           // Deciding which Position
           // Position - Belt
           IF "gtyp_Setup".i_Pos_Selection = 21 THEN
               #ldi_Pos_Horizontal := "gtyp_HBW".di_PosBelt_Horizontal;
               #ldi_Pos_Vertical := "gtyp_HBW".di_PosBelt_Vertical;
               #ldi_Offset_Vertical := "gtyp_HBW".di_Offset_Pos_Belt_Vertical;
               // Position - A1 
           ELSIF "gtyp_Setup".i_Pos_Selection = 22 THEN
               #ldi_Pos_Horizontal := "gtyp_HBW".di_PosRack_A1_Horizontal;
               #ldi_Pos_Vertical := "gtyp_HBW".di_PosRack_A1_Vertical;
               #ldi_Offset_Vertical := "gtyp_HBW".di_Offset_Pos_Rack_Vertical;
               // Position - B2 
           ELSIF "gtyp_Setup".i_Pos_Selection = 23 THEN
               #ldi_Pos_Horizontal := "gtyp_HBW".di_PosRack_B2_Horizontal;
               #ldi_Pos_Vertical := "gtyp_HBW".di_PosRack_B2_Vertical;
               #ldi_Offset_Vertical := "gtyp_HBW".di_Offset_Pos_Rack_Vertical;
               // Position - C3 
           ELSIF "gtyp_Setup".i_Pos_Selection = 24 THEN
               #ldi_Pos_Horizontal := "gtyp_HBW".di_PosRack_C3_Horizontal;
               #ldi_Pos_Vertical := "gtyp_HBW".di_PosRack_C3_Vertical;
               #ldi_Offset_Vertical := "gtyp_HBW".di_Offset_Pos_Rack_Vertical;
           END_IF;
       END_IF;

       // Set Positioning activ?
       IF NOT "gtyp_Setup".x_Set_Pos_Activ THEN
           "gtyp_Setup".i_Pos_Selection := 0;
       END_IF;

       // step chain HBW
       CASE #li_StepCase OF

           0:  // init
               #lx_Start_TON_Wait := FALSE;
               #li_StepCase := 10;

           10:  // Set Positioning activ?
               IF "gtyp_Setup".x_Set_Pos_Activ
                   AND (("gtyp_Setup".i_Pos_Selection > 20)
                   AND ("gtyp_Setup".i_Pos_Selection < 41)) THEN

                   "gtyp_HBW".Horizontal_Axis.x_Start_Positioning := FALSE;
                   "gtyp_HBW".Vertical_Axis.x_Start_Positioning := FALSE;
                   "gtyp_HBW".Horizontal_Axis.x_Reference := FALSE;
                   "gtyp_HBW".Vertical_Axis.x_Reference := FALSE;
                   "gtyp_Setup".x_Start_Positioning := FALSE;
                   "gtyp_Setup".x_Final_Positioning := FALSE;
                   "gtyp_Setup".x_Home_Positioning := FALSE;
                   "gtyp_Setup".x_Start_Offset := FALSE;
                   "QX_HBW_M4_CantileverBackward_Q8" := FALSE;
                   "QX_HBW_M4_CantileverForward_Q7" := FALSE;
                   #li_StepCase := 20;
               END_IF;

           20: //homing vertical/horizontal axis

               "gtyp_HBW".Horizontal_Axis.x_Reference := TRUE;
               "gtyp_HBW".Vertical_Axis.x_Reference := TRUE;

               IF NOT "gtyp_HBW".Horizontal_Axis.x_Referenced AND NOT "gtyp_HBW".Vertical_Axis.x_Referenced THEN
                   #li_StepCase := 30;
               END_IF;

           30: // homed vertical/horizontal axis
               IF "gtyp_HBW".Horizontal_Axis.x_Referenced THEN
                   "gtyp_HBW".Horizontal_Axis.x_Reference := FALSE;
               END_IF;
               IF "gtyp_HBW".Vertical_Axis.x_Referenced THEN
                   "gtyp_HBW".Vertical_Axis.x_Reference := FALSE;
               END_IF;

               IF "gtyp_HBW".Horizontal_Axis.x_Referenced AND "gtyp_HBW".Vertical_Axis.x_Referenced THEN
                   "gtyp_HBW".Horizontal_Axis.x_Reference := FALSE;
                   "gtyp_HBW".Vertical_Axis.x_Reference := FALSE;
                   #li_StepCase := 40;
               END_IF;

           40: // Start Positioning Step next
               IF "gtyp_Setup".x_Start_Positioning OR #lx_Start_Positioning_m OR #lx_Start_FinalPositioning_m OR #lx_Start_Offset_m THEN
                   #lx_Start_Positioning_m := FALSE;
                   #li_StepCase := 50;
               END_IF;

           50: // Position vertical/horizontal HBW
               "gtyp_HBW".Horizontal_Axis.di_Target_Position := #ldi_Pos_Horizontal;
               "gtyp_HBW".Horizontal_Axis.x_Start_Positioning := TRUE;
               "gtyp_HBW".Vertical_Axis.di_Target_Position := #ldi_Pos_Vertical;
               "gtyp_HBW".Vertical_Axis.x_Start_Positioning := TRUE;

               IF ("gtyp_HBW".Horizontal_Axis.di_Actual_Position <= (#ldi_Pos_Horizontal + "gtyp_HBW".Horizontal_Axis.Config.di_Pos_Window))
                   AND ("gtyp_HBW".Horizontal_Axis.di_Actual_Position >= (#ldi_Pos_Horizontal - "gtyp_HBW".Horizontal_Axis.Config.di_Pos_Window))
                   AND "gtyp_HBW".Horizontal_Axis.x_Position_Reached THEN
                   "gtyp_HBW".Horizontal_Axis.x_Start_Positioning := FALSE;
               END_IF;

               IF ("gtyp_HBW".Vertical_Axis.di_Actual_Position <= (#ldi_Pos_Vertical + "gtyp_HBW".Vertical_Axis.Config.di_Pos_Window))
                   AND ("gtyp_HBW".Vertical_Axis.di_Actual_Position >= (#ldi_Pos_Vertical - "gtyp_HBW".Vertical_Axis.Config.di_Pos_Window))
                   AND "gtyp_HBW".Vertical_Axis.x_Position_Reached THEN
                   "gtyp_HBW".Vertical_Axis.x_Start_Positioning := FALSE;
               END_IF;

               IF ("gtyp_HBW".Horizontal_Axis.di_Actual_Position <= (#ldi_Pos_Horizontal + "gtyp_HBW".Horizontal_Axis.Config.di_Pos_Window))
                   AND ("gtyp_HBW".Horizontal_Axis.di_Actual_Position >= (#ldi_Pos_Horizontal - "gtyp_HBW".Horizontal_Axis.Config.di_Pos_Window))
                   AND "gtyp_HBW".Horizontal_Axis.x_Position_Reached
                   AND ("gtyp_HBW".Vertical_Axis.di_Actual_Position <= (#ldi_Pos_Vertical + "gtyp_HBW".Vertical_Axis.Config.di_Pos_Window))
                   AND ("gtyp_HBW".Vertical_Axis.di_Actual_Position >= (#ldi_Pos_Vertical - "gtyp_HBW".Vertical_Axis.Config.di_Pos_Window))
                   AND "gtyp_HBW".Vertical_Axis.x_Position_Reached THEN
                   "gtyp_HBW".Horizontal_Axis.x_Start_Positioning := FALSE;
                   "gtyp_HBW".Vertical_Axis.x_Start_Positioning := FALSE;
                   "gtyp_Setup".x_Start_Positioning := FALSE;
                   #li_StepCase := 60;
               END_IF;

           60: // Deciding which doing

               // Start new Positioning
               IF "gtyp_Setup".x_Start_Positioning THEN
                   #lx_Start_Positioning_m := TRUE;
                   #li_StepCase := 10;
                   // Start Final Positioning
               ELSIF "gtyp_Setup".x_Final_Positioning OR #lx_Start_FinalPositioning_m OR #lx_Start_Offset_m THEN
                   #lx_Start_FinalPositioning_m := FALSE;
                   #li_StepCase := 70;
                   // Deaktivate Set Positioning
               ELSIF #lfb_R_Trig_Deaktivate.Q OR "gtyp_Setup".x_Home_Positioning THEN
                   "gtyp_Setup".x_Home_Positioning := FALSE;
                   #li_StepCase := 110;
               END_IF;

           70: // Final Positioning - Cantilever Forward

               "QX_HBW_M4_CantileverBackward_Q8" := FALSE;
               "QX_HBW_M4_CantileverForward_Q7" := TRUE;

               IF "IX_HBW_SwitchCantileverFront_I5" AND NOT "IX_HBW_SwitchCantileverBack_I6" THEN
                   "QX_HBW_M4_CantileverBackward_Q8" := FALSE;
                   "QX_HBW_M4_CantileverForward_Q7" := FALSE;
                   "gtyp_Setup".x_Final_Positioning := FALSE;
                   #li_StepCase := 80;
               END_IF;

           80: // Deciding which doing

               // Start new Positioning
               IF "gtyp_Setup".x_Start_Positioning THEN
                   #lx_Start_Positioning_m := TRUE;
                   #li_StepCase := 110;
                   // Start Final Positioning
               ELSIF "gtyp_Setup".x_Final_Positioning THEN
                   #lx_Start_FinalPositioning_m := TRUE;
                   #li_StepCase := 110;
                   // Start Final Positioning
               ELSIF "gtyp_Setup".x_Start_Offset OR #lx_Start_Offset_m THEN
                   #lx_Start_Offset_m := FALSE;
                   #li_StepCase := 90;
                   // Deaktivate Set Positioning
               ELSIF #lfb_R_Trig_Deaktivate.Q OR "gtyp_Setup".x_Home_Positioning THEN
                   "gtyp_Setup".x_Home_Positioning := FALSE;
                   #li_StepCase := 110;
               END_IF;

           90: // Position vertical+offset HBW
               "gtyp_HBW".Vertical_Axis.di_Target_Position := #ldi_Pos_Vertical - #ldi_Offset_Vertical;
               "gtyp_HBW".Vertical_Axis.x_Start_Positioning := TRUE;

               IF ("gtyp_HBW".Vertical_Axis.di_Actual_Position <= (#ldi_Pos_Vertical - #ldi_Offset_Vertical + "gtyp_HBW".Vertical_Axis.Config.di_Pos_Window))
                   AND ("gtyp_HBW".Vertical_Axis.di_Actual_Position >= (#ldi_Pos_Vertical - #ldi_Offset_Vertical - "gtyp_HBW".Vertical_Axis.Config.di_Pos_Window))
                   AND "gtyp_HBW".Vertical_Axis.x_Position_Reached THEN
                   "gtyp_HBW".Vertical_Axis.x_Start_Positioning := FALSE;
                   "gtyp_Setup".x_Start_Offset := FALSE;
                   #li_StepCase := 100;
               END_IF;

           100: // Deciding which doing

               // Start new Positioning
               IF "gtyp_Setup".x_Start_Positioning THEN
                   #lx_Start_Positioning_m := TRUE;
                   #li_StepCase := 110;
                   // Start Final Positioning
               ELSIF "gtyp_Setup".x_Final_Positioning THEN
                   #lx_Start_FinalPositioning_m := TRUE;
                   #li_StepCase := 110;
                   // Start Final Positioning
               ELSIF "gtyp_Setup".x_Start_Offset THEN
                   #lx_Start_Offset_m := true;
                   #li_StepCase := 110;
                   // Deaktivate Set Positioning
               ELSIF #lfb_R_Trig_Deaktivate.Q OR "gtyp_Setup".x_Home_Positioning THEN
                   "gtyp_Setup".x_Home_Positioning := FALSE;
                   #li_StepCase := 110;
               END_IF;

           110: // Position vertical HBW
               "gtyp_HBW".Vertical_Axis.di_Target_Position := #ldi_Pos_Vertical;
               "gtyp_HBW".Vertical_Axis.x_Start_Positioning := TRUE;

               IF ("gtyp_HBW".Vertical_Axis.di_Actual_Position <= (#ldi_Pos_Vertical + "gtyp_HBW".Vertical_Axis.Config.di_Pos_Window))
                   AND ("gtyp_HBW".Vertical_Axis.di_Actual_Position >= (#ldi_Pos_Vertical - "gtyp_HBW".Vertical_Axis.Config.di_Pos_Window))
                   AND "gtyp_HBW".Vertical_Axis.x_Position_Reached THEN
                   "gtyp_HBW".Vertical_Axis.x_Start_Positioning := FALSE;
                   #li_StepCase := 120;
               END_IF;

           120: // Position vertical Back HBW

               "QX_HBW_M4_CantileverBackward_Q8" := TRUE;
               "QX_HBW_M4_CantileverForward_Q7" := FALSE;

               IF NOT "IX_HBW_SwitchCantileverFront_I5" AND "IX_HBW_SwitchCantileverBack_I6" THEN
                   "QX_HBW_M4_CantileverBackward_Q8" := FALSE;
                   "QX_HBW_M4_CantileverForward_Q7" := FALSE;
                   #li_StepCase := 130;
               END_IF;

           130: // homing vertical/horizontal axis

               "gtyp_HBW".Horizontal_Axis.x_Reference := TRUE;
               "gtyp_HBW".Vertical_Axis.x_Reference := TRUE;

               IF NOT "gtyp_HBW".Horizontal_Axis.x_Referenced AND NOT "gtyp_HBW".Vertical_Axis.x_Referenced THEN
                   #li_StepCase := 140;
               END_IF;

           140: //homed vertical/horizontal axis
               IF "gtyp_HBW".Horizontal_Axis.x_Referenced THEN
                   "gtyp_HBW".Horizontal_Axis.x_Reference := FALSE;
               END_IF;
               IF "gtyp_HBW".Vertical_Axis.x_Referenced THEN
                   "gtyp_HBW".Vertical_Axis.x_Reference := FALSE;
               END_IF;

               IF "gtyp_HBW".Horizontal_Axis.x_Referenced AND "gtyp_HBW".Vertical_Axis.x_Referenced THEN
                   "gtyp_HBW".Horizontal_Axis.x_Reference := FALSE;
                   "gtyp_HBW".Vertical_Axis.x_Reference := FALSE;
                   #li_StepCase := 0;
               END_IF;

               // Statement section ELSE    
           ELSE
               ;
       END_CASE;

       IF (("gtyp_Setup".i_Pos_Selection > 20)
           AND ("gtyp_Setup".i_Pos_Selection < 41)) THEN
           // Reload Pos Value
           "gtyp_Setup".di_Pos_Horizontal := #ldi_Pos_Horizontal;
           "gtyp_Setup".di_Pos_Vertical := #ldi_Pos_Vertical;
           "gtyp_Setup".di_Pos_Rotate := 0;
       END_IF;
   ELSE
       #lx_Init := TRUE;
   END_IF;
END_FUNCTION_BLOCK

FUNCTION_BLOCK "PRG_SSC_Calibration_Color"   // FB32, SCL
TITLE = Program Calibration Color Sensor SSC
{ S7_Optimized_Access := 'TRUE' }
AUTHOR : A.Schaefer
VERSION : 0.0
   VAR
      lx_Init : Bool;
      lx_Start_TON_Wait : Bool;
      lx_Start_Positioning_m : Bool;
      lt_TON_Wait : Time;
      li_StepCase : Int;
      ldi_Pos_Horizontal : DInt;
      ldi_Pos_Vertical : DInt;
      lfb_R_Trig_Deaktivate : R_TRIG;
      lfb_TON_Wait : TON_TIME;
   END_VAR
BEGIN
   IF #lx_Init THEN

       // FB TON Wait
       #lfb_TON_Wait(IN := #lx_Start_TON_Wait,
                     PT := #lt_TON_Wait);

       #lfb_R_Trig_Deaktivate(CLK := NOT "gtyp_Setup".x_Color_Sensor_Calibration
                              OR NOT ("gtyp_Setup".i_Color_Sensor_Selection = 1));
       // Deaktivate step 0   
       IF #lfb_R_Trig_Deaktivate.Q THEN
           "gtyp_Setup".x_Calculate_Value_Color := FALSE;
           "gtyp_Setup".x_Set_Calib_Value_Color_Blue := FALSE;
           "gtyp_Setup".x_Set_Calib_Value_Color_Red := FALSE;
           "gtyp_Setup".x_Set_Calib_Value_Color_White := FALSE;
           "gtyp_Setup".w_Calib_ColorValue_Blue := 0;
           "gtyp_Setup".w_Calib_ColorValue_Red := 0;
           "gtyp_Setup".w_Calib_ColorValue_White := 0;
           "gtyp_Setup".w_Threshold_Red_Blue := 0;
           "gtyp_Setup".w_Threshold_White_Red := 0;
           #li_StepCase := 0;
       END_IF;

       // step chain HBW
       CASE #li_StepCase OF

           0:  // init
               #lx_Start_TON_Wait := FALSE;
               #li_StepCase := 10;

           10:  // Set Calibration activ?
               IF "gtyp_Setup".x_Color_Sensor_Calibration
                   AND ("gtyp_Setup".i_Color_Sensor_Selection = 1) THEN
                   "gtyp_Setup".x_Calculate_Value_Color := FALSE;
                   "gtyp_Setup".x_Set_Calib_Value_Color_Blue := FALSE;
                   "gtyp_Setup".x_Set_Calib_Value_Color_Red := FALSE;
                   "gtyp_Setup".x_Set_Calib_Value_Color_White := FALSE;
                   "gtyp_Setup".w_Calib_ColorValue_Blue := 0;
                   "gtyp_Setup".w_Calib_ColorValue_Red := 0;
                   "gtyp_Setup".w_Calib_ColorValue_White := 0;
                   "gtyp_Setup".w_Threshold_Red_Blue := 0;
                   "gtyp_Setup".w_Threshold_White_Red := 0;
                   #li_StepCase := 20;
               END_IF;

           20: // wait for set Values or Calculate

               // Start new Positioning
               IF "gtyp_Setup".x_Set_Calib_Value_Color_Blue THEN
                   "gtyp_Setup".w_Calib_ColorValue_Blue := "IW_SSC_ColorSensor_A1";
                   "gtyp_Setup".x_Set_Calib_Value_Color_Blue := FALSE;
               ELSIF "gtyp_Setup".x_Set_Calib_Value_Color_Red THEN
                   "gtyp_Setup".w_Calib_ColorValue_Red := "IW_SSC_ColorSensor_A1";
                   "gtyp_Setup".x_Set_Calib_Value_Color_Red := FALSE;
               ELSIF "gtyp_Setup".x_Set_Calib_Value_Color_White THEN
                   "gtyp_Setup".w_Calib_ColorValue_White := "IW_SSC_ColorSensor_A1";
                   "gtyp_Setup".x_Set_Calib_Value_Color_White := FALSE;
               END_IF;

               "gtyp_Setup".w_Threshold_White_Red := "gtyp_Setup".w_Calib_ColorValue_White + (("gtyp_Setup".w_Calib_ColorValue_Red - "gtyp_Setup".w_Calib_ColorValue_White) / 2);
               "gtyp_Setup".w_Threshold_Red_Blue := "gtyp_Setup".w_Calib_ColorValue_Red + (("gtyp_Setup".w_Calib_ColorValue_Blue - "gtyp_Setup".w_Calib_ColorValue_Red) / 2);

               IF "gtyp_Setup".x_Calculate_Value_Color THEN
                   "gtyp_SSC".w_Threshold_White_Red := "gtyp_Setup".w_Threshold_White_Red;
                   "gtyp_SSC".w_Threshold_Red_Blue := "gtyp_Setup".w_Threshold_Red_Blue;
                   "gtyp_Setup".x_Calculate_Value_Color := FALSE;
               END_IF;

               // Statement section ELSE    
           ELSE
               ;
       END_CASE;

       IF ("gtyp_Setup".i_Color_Sensor_Selection = 1) THEN
           // Reload Pos Value
           "gtyp_Setup".w_Actual_ColorValue := "IW_SSC_ColorSensor_A1";
       END_IF;
   ELSE
       #lx_Init := TRUE;
   END_IF;
END_FUNCTION_BLOCK

FUNCTION_BLOCK "PRG_SLD_Calibration_Color"   // FB33, SCL
TITLE = Program Calibration Color Sensor SLD
{ S7_Optimized_Access := 'TRUE' }
AUTHOR : A.Schaefer
VERSION : 0.0
   VAR
      lx_Init : Bool;
      lx_Start_TON_Wait : Bool;
      lx_Start_Positioning_m : Bool;
      lt_TON_Wait : Time;
      li_StepCase : Int;
      lw_ColorValueMin : Word;
      ldi_Pos_Horizontal : DInt;
      ldi_Pos_Vertical : DInt;
      lfb_R_Trig_Deaktivate : R_TRIG;
      lfb_TON_Wait : TON_TIME;
   END_VAR
BEGIN
   IF #lx_Init THEN

       // FB TON Wait
       #lfb_TON_Wait(IN := #lx_Start_TON_Wait,
                     PT := #lt_TON_Wait);

       #lfb_R_Trig_Deaktivate(CLK := NOT "gtyp_Setup".x_Color_Sensor_Calibration
                              OR NOT ("gtyp_Setup".i_Color_Sensor_Selection = 2));
       // Deaktivate step 0   
       IF #lfb_R_Trig_Deaktivate.Q THEN
           "gtyp_Setup".x_Calculate_Value_Color := FALSE;
           "gtyp_Setup".x_Set_Calib_Value_Color_Blue := FALSE;
           "gtyp_Setup".x_Set_Calib_Value_Color_Red := FALSE;
           "gtyp_Setup".x_Set_Calib_Value_Color_White := FALSE;
           "gtyp_Setup".w_Calib_ColorValue_Blue := 0;
           "gtyp_Setup".w_Calib_ColorValue_Red := 0;
           "gtyp_Setup".w_Calib_ColorValue_White := 0;
           "gtyp_Setup".w_Threshold_Red_Blue := 0;
           "gtyp_Setup".w_Threshold_White_Red := 0;
           "QX_SLD_M1_ConveyorBelt_Q1" := FALSE;
           #lw_ColorValueMin := 16#FF;
           #li_StepCase := 0;
       END_IF;

       // step chain HBW
       CASE #li_StepCase OF

           0:  // init
               #lx_Start_TON_Wait := FALSE;
               #li_StepCase := 10;

           10:  // Set Calibration activ?
               IF "gtyp_Setup".x_Color_Sensor_Calibration
                   AND ("gtyp_Setup".i_Color_Sensor_Selection = 2) THEN
                   "gtyp_Setup".x_Calculate_Value_Color := FALSE;
                   "gtyp_Setup".x_Set_Calib_Value_Color_Blue := FALSE;
                   "gtyp_Setup".x_Set_Calib_Value_Color_Red := FALSE;
                   "gtyp_Setup".x_Set_Calib_Value_Color_White := FALSE;
                   "gtyp_Setup".w_Calib_ColorValue_Blue := 0;
                   "gtyp_Setup".w_Calib_ColorValue_Red := 0;
                   "gtyp_Setup".w_Calib_ColorValue_White := 0;
                   "gtyp_Setup".w_Threshold_Red_Blue := 0;
                   "gtyp_Setup".w_Threshold_White_Red := 0;
                   "QX_SLD_M1_ConveyorBelt_Q1" := FALSE;
                   #lw_ColorValueMin := 16#FFFF;
                   #li_StepCase := 20;
               END_IF;

           20: // wait for set Values or Calculate

               IF NOT "IX_SLD_LightBarrierInlet_I2" THEN
                   "QX_SLD_M1_ConveyorBelt_Q1" := TRUE;
                   #lw_ColorValueMin := 16#FFFF;
               END_IF;

               IF #lw_ColorValueMin > "IW_SLD_ColorSensor_A4" THEN
                   #lw_ColorValueMin := "IW_SLD_ColorSensor_A4";
               END_IF;

               IF NOT "IX_SLD_LightBarrierBehindColorSensor_I3" THEN
                   "QX_SLD_M1_ConveyorBelt_Q1" := FALSE;
               END_IF;

               // Start new Positioning
               IF "gtyp_Setup".x_Set_Calib_Value_Color_Blue THEN
                   "gtyp_Setup".w_Calib_ColorValue_Blue := #lw_ColorValueMin;
                   "gtyp_Setup".x_Set_Calib_Value_Color_Blue := FALSE;
               ELSIF "gtyp_Setup".x_Set_Calib_Value_Color_Red THEN
                   "gtyp_Setup".w_Calib_ColorValue_Red := #lw_ColorValueMin;
                   "gtyp_Setup".x_Set_Calib_Value_Color_Red := FALSE;
               ELSIF "gtyp_Setup".x_Set_Calib_Value_Color_White THEN
                   "gtyp_Setup".w_Calib_ColorValue_White := #lw_ColorValueMin;
                   "gtyp_Setup".x_Set_Calib_Value_Color_White := FALSE;
               END_IF;

               "gtyp_Setup".w_Threshold_White_Red := "gtyp_Setup".w_Calib_ColorValue_White + (("gtyp_Setup".w_Calib_ColorValue_Red - "gtyp_Setup".w_Calib_ColorValue_White) / 2);
               "gtyp_Setup".w_Threshold_Red_Blue := "gtyp_Setup".w_Calib_ColorValue_Red + (("gtyp_Setup".w_Calib_ColorValue_Blue - "gtyp_Setup".w_Calib_ColorValue_Red) / 2);

               IF "gtyp_Setup".x_Calculate_Value_Color THEN
                   "gtyp_SLD".w_Threshold_White_Red := "gtyp_Setup".w_Threshold_White_Red;
                   "gtyp_SLD".w_Threshold_Red_Blue := "gtyp_Setup".w_Threshold_Red_Blue;
                   "gtyp_Setup".x_Calculate_Value_Color := FALSE;
               END_IF;

               // Statement section ELSE    
           ELSE
               ;
       END_CASE;

       IF ("gtyp_Setup".i_Color_Sensor_Selection = 2) THEN
           // Reload Pos Value
           "gtyp_Setup".w_Actual_ColorValue := "IW_SLD_ColorSensor_A4";
       END_IF;
   ELSE
       #lx_Init := TRUE;
   END_IF;
END_FUNCTION_BLOCK

FUNCTION_BLOCK "PRG_SLD_Set_Counter_Values"   // FB34, SCL
TITLE = Program Set counter Values SLD
{ S7_Optimized_Access := 'TRUE' }
AUTHOR : A.Schaefer
VERSION : 0.0
   VAR
      lx_Init : Bool;
      lfb_R_Trig_Calib_activ : R_TRIG;
   END_VAR
BEGIN
   IF #lx_Init THEN

       // Reload act. Counter Values
       IF NOT "gtyp_Setup".x_Counter_Value_Calibration THEN
           "gtyp_Setup".i_Calib_CounterValue_Blue := "gtyp_SLD".i_CounterValue_Blue;
           "gtyp_Setup".i_Calib_CounterValue_Red := "gtyp_SLD".i_CounterValue_Red;
           "gtyp_Setup".i_Calib_CounterValue_White := "gtyp_SLD".i_CounterValue_White;
       END_IF;

       // Set Counter Values   
       IF "gtyp_Setup".x_Set_CounterValues AND "gtyp_Setup".x_Counter_Value_Calibration THEN
           "gtyp_SLD".i_CounterValue_Blue := "gtyp_Setup".i_Calib_CounterValue_Blue;
           "gtyp_SLD".i_CounterValue_Red := "gtyp_Setup".i_Calib_CounterValue_Red;
           "gtyp_SLD".i_CounterValue_White := "gtyp_Setup".i_Calib_CounterValue_White;
           "gtyp_Setup".x_Set_CounterValues := FALSE;
       END_IF;

   ELSE
       #lx_Init := TRUE;
   END_IF;
END_FUNCTION_BLOCK

FUNCTION_BLOCK "PRG_VGR_Set_Park_Position"   // FB35, SCL
TITLE = Program Set Positioning VGR
{ S7_Optimized_Access := 'TRUE' }
AUTHOR : A.Schaefer
VERSION : 0.0
   VAR
      lx_Init : Bool;
      lx_Start_TON_Wait : Bool;
      lt_TON_Wait : Time;
      li_StepCase : Int;
      lfb_TON_Wait : TON_TIME;
      lfb_R_Trig_Start_Park_Pos : R_TRIG;
   END_VAR
BEGIN
   IF #lx_Init THEN

       // FB TON Wait
       #lfb_TON_Wait(IN := #lx_Start_TON_Wait,
                     PT := #lt_TON_Wait);

       #lfb_R_Trig_Start_Park_Pos(CLK := "gtyp_Setup".x_Park_Position
                                  OR "IX_Set_Park_Position");

       // Set Start Park Position   
       IF #lfb_R_Trig_Start_Park_Pos.Q THEN
           "gtyp_VGR".x_Start_Park_Position := TRUE;
           #li_StepCase := 0;
       END_IF;

       // not Start Park Pos Step 0
       IF NOT "gtyp_VGR".x_Start_Park_Position THEN
           #li_StepCase := 0;
       END_IF;

       // step chain HBW
       CASE #li_StepCase OF

           0:  // init
               #lx_Start_TON_Wait := FALSE;
               #li_StepCase := 10;

           10:  // Set Positioning activ?
               IF "gtyp_VGR".x_Start_Park_Position AND NOT "gtyp_VGR".x_Park_Position_Reached THEN
                   "gtyp_VGR".horizontal_Axis.x_Start_Positioning := FALSE;
                   "gtyp_VGR".vertical_Axis.x_Start_Positioning := FALSE;
                   "gtyp_VGR".rotate_Axis.x_Start_Positioning := FALSE;
                   "gtyp_VGR".horizontal_Axis.x_Reference := FALSE;
                   "gtyp_VGR".vertical_Axis.x_Reference := FALSE;
                   "gtyp_VGR".rotate_Axis.x_Reference := FALSE;
                   "gtyp_VGR".vertical_Axis.i_PWM := 800;
                   #li_StepCase := 20;
               END_IF;

           20: // homing vertical axis
               "gtyp_VGR".vertical_Axis.x_Reference := TRUE;

               IF NOT "gtyp_VGR".vertical_Axis.x_Referenced THEN
                   #li_StepCase := 30;
               END_IF;

           30: // homed vertical axis
               IF "gtyp_VGR".vertical_Axis.x_Referenced THEN
                   "gtyp_VGR".vertical_Axis.x_Reference := FALSE;
                   #li_StepCase := 40;
               END_IF;

           40: // homing horizontal axis
               "gtyp_VGR".horizontal_Axis.x_Reference := TRUE;

               IF NOT "gtyp_VGR".horizontal_Axis.x_Referenced THEN
                   #li_StepCase := 50;
               END_IF;

           50: // homed horizontal axis
               IF "gtyp_VGR".horizontal_Axis.x_Referenced THEN
                   "gtyp_VGR".horizontal_Axis.x_Reference := FALSE;
                   #li_StepCase := 60;
               END_IF;

           60: // homing rotate axis
               "gtyp_VGR".rotate_Axis.x_Reference := TRUE;

               IF NOT "gtyp_VGR".rotate_Axis.x_Referenced THEN
                   #li_StepCase := 70;
               END_IF;

           70: // homed rotate axis
               IF "gtyp_VGR".rotate_Axis.x_Referenced THEN
                   "gtyp_VGR".rotate_Axis.x_Reference := FALSE;
                   #li_StepCase := 80;
               END_IF;

           80: // Position rotate Axis
               "gtyp_VGR".rotate_Axis.di_Target_Position := "gtyp_VGR".di_Pos_Park_rotate;
               "gtyp_VGR".rotate_Axis.x_Start_Positioning := TRUE;

               IF ("gtyp_VGR".rotate_Axis.di_Actual_Position <= ("gtyp_VGR".di_Pos_Park_rotate + "gtyp_VGR".rotate_Axis.Config.di_Pos_Window))
                   AND ("gtyp_VGR".rotate_Axis.di_Actual_Position >= ("gtyp_VGR".di_Pos_Park_rotate - "gtyp_VGR".rotate_Axis.Config.di_Pos_Window))
                   AND "gtyp_VGR".rotate_Axis.x_Position_Reached THEN
                   "gtyp_VGR".rotate_Axis.x_Start_Positioning := FALSE;
                   #li_StepCase := 90;
               END_IF;

           90: // Position horizontal Axis
               "gtyp_VGR".horizontal_Axis.di_Target_Position := "gtyp_VGR".di_Pos_Park_horizontal;
               "gtyp_VGR".horizontal_Axis.x_Start_Positioning := TRUE;

               IF ("gtyp_VGR".horizontal_Axis.di_Actual_Position <= ("gtyp_VGR".di_Pos_Park_horizontal + "gtyp_VGR".horizontal_Axis.Config.di_Pos_Window))
                   AND ("gtyp_VGR".horizontal_Axis.di_Actual_Position >= ("gtyp_VGR".di_Pos_Park_horizontal - "gtyp_VGR".horizontal_Axis.Config.di_Pos_Window))
                   AND "gtyp_VGR".horizontal_Axis.x_Position_Reached THEN
                   "gtyp_VGR".horizontal_Axis.x_Start_Positioning := FALSE;
                   #li_StepCase := 100;
               END_IF;

           100: // Position vertical Axis
               "gtyp_VGR".vertical_Axis.i_PWM := 500;
               "gtyp_VGR".vertical_Axis.di_Target_Position := "gtyp_VGR".di_Pos_Park_vertical;
               "gtyp_VGR".vertical_Axis.x_Start_Positioning := TRUE;

               IF ("gtyp_VGR".vertical_Axis.di_Actual_Position <= ("gtyp_VGR".di_Pos_Park_vertical + "gtyp_VGR".vertical_Axis.Config.di_Pos_Window))
                   AND ("gtyp_VGR".vertical_Axis.di_Actual_Position >= ("gtyp_VGR".di_Pos_Park_vertical - "gtyp_VGR".vertical_Axis.Config.di_Pos_Window))
                   AND "gtyp_VGR".vertical_Axis.x_Position_Reached THEN
                   "gtyp_VGR".vertical_Axis.x_Start_Positioning := FALSE;
                   #li_StepCase := 110;
               END_IF;

           110: // Deciding which doing
               "gtyp_VGR".x_Park_Position_Reached := TRUE;


               // Statement section ELSE    
           ELSE
               ;
       END_CASE;

   ELSE
       #lx_Init := TRUE;
   END_IF;
END_FUNCTION_BLOCK

FUNCTION_BLOCK "PRG_DSO_Status"   // FB36, SCL
TITLE = Program Status DSO
{ S7_Optimized_Access := 'TRUE' }
AUTHOR : A.Schaefer
VERSION : 0.0
   VAR
      lx_Init : Bool;
      lx_Start : Bool;
      li_StepCase : Int;
      ldt_MQTT : Date_And_Time;
      li_Return_LDT : Int;
      li_code_old : Int;
      lfb_R_Trig_Outsourcing : R_TRIG;
      lfb_R_Trig_Take_Workpiece : R_TRIG;
      lfb_TON_Status : TON_TIME;
      lfb_TON_End_Order : TON_TIME;
      lx_StartStatus : Bool;
      lx_StartEndOrder : Bool;
      lx_StartTimer : Bool;
   END_VAR
BEGIN
   IF #lx_Init THEN

       // wait time state
       #lfb_TON_Status(IN := NOT #lx_StartStatus,
                       PT := T#2s);

       // rising/falling edge light barrier DSI
       #lfb_R_Trig_Outsourcing(CLK := NOT "IX_SSC_LightBarrierOutsourcing_I4");
       #lfb_R_Trig_Take_Workpiece(CLK := "IX_SSC_LightBarrierOutsourcing_I4");

       // start wait time end order 
       IF NOT "IX_SSC_LightBarrierOutsourcing_I4" AND ("gtyp_Interface_Dashboard".Subscribe.State_Order.s_state = 'SHIPPED') THEN
           #lx_StartEndOrder := TRUE;
       END_IF;

       // wait time end order
       #lfb_TON_End_Order(IN := #lx_StartEndOrder,
                          PT := T#5s);

       IF #lfb_R_Trig_Take_Workpiece.Q OR #lfb_TON_End_Order.Q THEN
           #lx_StartEndOrder := FALSE;
           "gtyp_Interface_Dashboard".Subscribe.State_Order.ldt_ts := DT_TO_LDT(#ldt_MQTT);
           "gtyp_Interface_Dashboard".Subscribe.State_Order.s_state := 'WAITING_FOR_ORDER';
           "gtyp_Interface_Dashboard".Subscribe.State_Order.s_type := '';
           "gtyp_Interface_Dashboard".Subscribe.State_DSO.x_active := FALSE;
       END_IF;

       // state of the DSO transmitted to the cloud
       IF (#lfb_TON_Status.Q OR #lfb_R_Trig_Outsourcing.Q OR #lfb_R_Trig_Take_Workpiece.Q) AND NOT #lx_StartStatus THEN
           #lx_StartStatus := TRUE;
           #li_Return_LDT := RD_SYS_T(#ldt_MQTT);
           IF NOT "IX_SSC_LightBarrierOutsourcing_I4" THEN
               "gtyp_Interface_Dashboard".Subscribe.State_DSO.i_code := 0;
           ELSE
               "gtyp_Interface_Dashboard".Subscribe.State_DSO.i_code := 1;
           END_IF;
           "gtyp_Interface_Dashboard".Subscribe.State_DSO.ldt_ts := DT_TO_LDT(#ldt_MQTT);
           "gtyp_Interface_Dashboard".Subscribe.State_DSO.s_station := 'dso';
           "gtyp_Interface_Dashboard".Subscribe.State_DSO.s_target := '';
           "gtyp_Interface_Dashboard".Subscribe.State_DSO.s_description := '';
       END_IF;

       IF NOT #lfb_TON_Status.Q AND #lx_StartStatus THEN
           #lx_StartStatus := FALSE;
       END_IF;
   ELSE
       #lx_Init := TRUE;
       #lx_StartEndOrder := FALSE;
   END_IF;
END_FUNCTION_BLOCK

FUNCTION_BLOCK "PRG_DSI_Status"   // FB37, SCL
TITLE = Program Status DSI
{ S7_Optimized_Access := 'TRUE' }
AUTHOR : A.Schaefer
VERSION : 0.0
   VAR
      lx_Init : Bool;
      lx_Start : Bool;
      li_StepCase : Int;
      ldt_MQTT : Date_And_Time;
      li_Return_LDT : Int;
      lfb_R_Trig_Storage : R_TRIG;
      lfb_F_Trig_Storage : F_TRIG;
      lfb_TON_Status : TON_TIME;
      lx_StartStatus : Bool;
      lfb_TON_Schritt : TON_TIME;
      lx_StartTimer : Bool;
   END_VAR
BEGIN
   IF #lx_Init THEN

       // wait time state
       #lfb_TON_Status(IN := NOT #lx_StartStatus,
                       PT := T#2s);

       // rising/falling edge light barrier DSI
       #lfb_R_Trig_Storage(CLK := NOT "IX_SSC_LightBarrierStorage_I3");
       #lfb_F_Trig_Storage(CLK := NOT "IX_SSC_LightBarrierStorage_I3");

       // state of the DSI transmitted to the cloud
       IF (#lfb_TON_Status.Q OR #lfb_R_Trig_Storage.Q OR #lfb_F_Trig_Storage.Q) AND NOT #lx_StartStatus THEN
           #lx_StartStatus := TRUE;
           #li_Return_LDT := RD_SYS_T(#ldt_MQTT);
           IF NOT "IX_SSC_LightBarrierStorage_I3" THEN
               "gtyp_Interface_Dashboard".Subscribe.State_DSI.i_code := 0;
               "gtyp_Interface_Dashboard".Subscribe.State_DSI.x_active := TRUE;
           ELSE
               "gtyp_Interface_Dashboard".Subscribe.State_DSI.i_code := 1;
               IF #lfb_F_Trig_Storage.Q THEN
                   "gtyp_Interface_Dashboard".Subscribe.State_DSI.x_active := FALSE;
               END_IF;
           END_IF;
           "gtyp_Interface_Dashboard".Subscribe.State_DSI.ldt_ts := DT_TO_LDT(#ldt_MQTT);
           "gtyp_Interface_Dashboard".Subscribe.State_DSI.s_station := 'dsi';
           "gtyp_Interface_Dashboard".Subscribe.State_DSI.s_target := '';
           "gtyp_Interface_Dashboard".Subscribe.State_DSI.s_description := '';
       END_IF;

       IF NOT #lfb_TON_Status.Q AND #lx_StartStatus THEN
           #lx_StartStatus := FALSE;
       END_IF;
   ELSE
       #lx_Init := TRUE;
   END_IF;
END_FUNCTION_BLOCK

FUNCTION_BLOCK "PRG_SSC_Set_Park_Position"   // FB38, SCL
TITLE = Program Set Positioning SSC
{ S7_Optimized_Access := 'TRUE' }
AUTHOR : A.Schaefer
VERSION : 0.0
   VAR
      lx_Init : Bool;
      lx_Start_TON_Wait : Bool;
      lt_TON_Wait : Time;
      li_StepCase : Int;
      lfb_TON_Wait : TON_TIME;
      lfb_R_Trig_Start_Park_Pos : R_TRIG;
   END_VAR
BEGIN
   IF #lx_Init THEN

       // FB TON Wait
       #lfb_TON_Wait(IN := #lx_Start_TON_Wait,
                     PT := #lt_TON_Wait);

       #lfb_R_Trig_Start_Park_Pos(CLK := "gtyp_Setup".x_Park_Position
                                  OR "IX_Set_Park_Position");

       // Set Start Park Position   
       IF #lfb_R_Trig_Start_Park_Pos.Q THEN
           "gtyp_SSC".x_Start_Park_Position := TRUE;
           #li_StepCase := 0;
       END_IF;

       // not Start Park Pos Step 0
       IF NOT "gtyp_SSC".x_Start_Park_Position THEN
           #li_StepCase := 0;
       END_IF;

       // step chain HBW
       CASE #li_StepCase OF

           0:  // init
               #lx_Start_TON_Wait := FALSE;
               #li_StepCase := 10;

           10:  // Set Positioning activ?
               IF "gtyp_SSC".x_Start_Park_Position AND NOT "gtyp_SSC".x_Park_Position_Reached THEN
                   "gtyp_SSC".Horizontal_Axis.x_Start_Positioning := FALSE;
                   "gtyp_SSC".Vertical_Axis.x_Start_Positioning := FALSE;
                   "gtyp_SSC".Horizontal_Axis.x_Reference := FALSE;
                   "gtyp_SSC".Vertical_Axis.x_Reference := FALSE;
                   #li_StepCase := 20;
               END_IF;

           20: // homing vertical axis
               "gtyp_SSC".Vertical_Axis.x_Reference := TRUE;

               IF NOT "gtyp_SSC".Vertical_Axis.x_Referenced THEN
                   #li_StepCase := 30;
               END_IF;

           30: // homed vertical axis
               IF "gtyp_SSC".Vertical_Axis.x_Referenced THEN
                   "gtyp_SSC".Vertical_Axis.x_Reference := FALSE;
                   #li_StepCase := 40;
               END_IF;

           40: // homing horizontal axis
               "gtyp_SSC".Horizontal_Axis.x_Reference := TRUE;

               IF NOT "gtyp_SSC".Horizontal_Axis.x_Referenced THEN
                   #li_StepCase := 50;
               END_IF;

           50: // homed horizontal axis
               IF "gtyp_SSC".Horizontal_Axis.x_Referenced THEN
                   "gtyp_SSC".Horizontal_Axis.x_Reference := FALSE;
                   #li_StepCase := 60;
               END_IF;

           60: // Position horizontal Axis
               "gtyp_SSC".Horizontal_Axis.di_Target_Position := "gtyp_SSC".di_Pos_Park_Horizontal;
               "gtyp_SSC".Horizontal_Axis.x_Start_Positioning := TRUE;

               IF ("gtyp_SSC".Horizontal_Axis.di_Actual_Position <= ("gtyp_SSC".di_Pos_Park_Horizontal + "gtyp_SSC".Horizontal_Axis.Config.di_Pos_Window))
                   AND ("gtyp_SSC".Horizontal_Axis.di_Actual_Position >= ("gtyp_SSC".di_Pos_Park_Horizontal - "gtyp_SSC".Horizontal_Axis.Config.di_Pos_Window))
                   AND "gtyp_SSC".Horizontal_Axis.x_Position_Reached THEN
                   "gtyp_SSC".Horizontal_Axis.x_Start_Positioning := FALSE;
                   #li_StepCase := 70;
               END_IF;

           70: // Position vertical Axis
               "gtyp_SSC".Vertical_Axis.di_Target_Position := "gtyp_SSC".di_Pos_Park_Vertical;
               "gtyp_SSC".Vertical_Axis.x_Start_Positioning := TRUE;

               IF ("gtyp_SSC".Vertical_Axis.di_Actual_Position <= ("gtyp_SSC".di_Pos_Park_Vertical + "gtyp_SSC".Vertical_Axis.Config.di_Pos_Window))
                   AND ("gtyp_SSC".Vertical_Axis.di_Actual_Position >= ("gtyp_SSC".di_Pos_Park_Vertical - "gtyp_SSC".Vertical_Axis.Config.di_Pos_Window))
                   AND "gtyp_SSC".Vertical_Axis.x_Position_Reached THEN
                   "gtyp_SSC".Vertical_Axis.x_Start_Positioning := FALSE;
                   #li_StepCase := 80;
               END_IF;

           80: // Deciding which doing
               "gtyp_SSC".x_Park_Position_Reached := TRUE;


               // Statement section ELSE    
           ELSE
               ;
       END_CASE;

   ELSE
       #lx_Init := TRUE;
   END_IF;
END_FUNCTION_BLOCK

FUNCTION_BLOCK "PRG_MPO_Set_Park_Position"   // FB39, SCL
TITLE = Program Set Positioning HBW
{ S7_Optimized_Access := 'TRUE' }
AUTHOR : A.Schaefer
VERSION : 0.0
   VAR
      lx_Init : Bool;
      lx_Start_TON_Wait : Bool;
      lt_TON_Wait : Time;
      li_StepCase : Int;
      lfb_TON_Wait : TON_TIME;
      lfb_R_Trig_Start_Park_Pos : R_TRIG;
   END_VAR
BEGIN
   IF #lx_Init THEN

       // FB TON Wait
       #lfb_TON_Wait(IN := #lx_Start_TON_Wait,
                     PT := #lt_TON_Wait);

       #lfb_R_Trig_Start_Park_Pos(CLK := "gtyp_Setup".x_Park_Position
                                  OR "IX_Set_Park_Position");

       // Set Start Park Position   
       IF #lfb_R_Trig_Start_Park_Pos.Q THEN
           "gtyp_MPO".x_Start_Park_Position := TRUE;
           #li_StepCase := 0;
       END_IF;

       // not Start Park Pos Step 0
       IF NOT "gtyp_MPO".x_Start_Park_Position THEN
           #li_StepCase := 0;
       END_IF;

       // step chain HBW
       CASE #li_StepCase OF

           0:  // init
               #lx_Start_TON_Wait := FALSE;
               #li_StepCase := 10;

           10:  // Set Positioning activ?
               IF "gtyp_MPO".x_Start_Park_Position AND NOT "gtyp_MPO".x_Park_Position_Reached THEN
                   #li_StepCase := 20;
               END_IF;

           20: // Towards
               "QX_MPO_M5_VacuumTowardsTurnTable_Q8" := FALSE;
               "QX_MPO_M5_VacuumTowardsOven_Q7" := TRUE;
               #lx_Start_TON_Wait := TRUE;
               #lt_TON_Wait := T#4000ms;

               IF #lfb_TON_Wait.Q THEN
                   "QX_MPO_M5_VacuumTowardsTurnTable_Q8" := FALSE;
                   "QX_MPO_M5_VacuumTowardsOven_Q7" := FALSE;
                   #lx_Start_TON_Wait := FALSE;
                   #li_StepCase := 30;
               END_IF;

           30: // homing vertical axis
               "QX_MPO_M1_TurnTableClockwise_Q1" := TRUE;
               "QX_MPO_M1_TurnTableCounterclockwise_Q2" := FALSE;
               #lx_Start_TON_Wait := TRUE;
               #lt_TON_Wait := T#1000ms;

               IF #lfb_TON_Wait.Q THEN
                   "QX_MPO_M1_TurnTableClockwise_Q1" := FALSE;
                   "QX_MPO_M1_TurnTableCounterclockwise_Q2" := FALSE;
                   #lx_Start_TON_Wait := FALSE;
                   #li_StepCase := 40;
               END_IF;

           40: // Deciding which doing
               "gtyp_MPO".x_Park_Position_Reached := TRUE;


               // Statement section ELSE    
           ELSE
               ;
       END_CASE;

   ELSE
       #lx_Init := TRUE;
   END_IF;
END_FUNCTION_BLOCK

FUNCTION_BLOCK "PRG_HBW_Set_Park_Position"   // FB40, SCL
TITLE = Program Set Positioning HBW
{ S7_Optimized_Access := 'TRUE' }
AUTHOR : A.Schaefer
VERSION : 0.0
   VAR
      lx_Init : Bool;
      lx_Start_TON_Wait : Bool;
      lt_TON_Wait : Time;
      li_StepCase : Int;
      lfb_TON_Wait : TON_TIME;
      lfb_R_Trig_Start_Park_Pos : R_TRIG;
   END_VAR
BEGIN
   IF #lx_Init THEN

       // FB TON Wait
       #lfb_TON_Wait(IN := #lx_Start_TON_Wait,
                     PT := #lt_TON_Wait);

       #lfb_R_Trig_Start_Park_Pos(CLK := "gtyp_Setup".x_Park_Position
                                  OR "IX_Set_Park_Position");

       // Set Start Park Position   
       IF #lfb_R_Trig_Start_Park_Pos.Q THEN
           "gtyp_HBW".x_Start_Park_Position := TRUE;
           #li_StepCase := 0;
       END_IF;

       // not Start Park Pos Step 0
       IF NOT "gtyp_HBW".x_Start_Park_Position THEN
           #li_StepCase := 0;
       END_IF;

       // step chain HBW
       CASE #li_StepCase OF

           0:  // init
               #lx_Start_TON_Wait := FALSE;
               #li_StepCase := 10;

           10:  // Set Positioning activ?
               IF "IX_HBW_SwitchCantileverFront_I5" OR NOT "IX_HBW_SwitchCantileverBack_I6" THEN
                   "QX_HBW_M4_CantileverBackward_Q8" := TRUE;
                   "QX_HBW_M4_CantileverForward_Q7" := FALSE;
               ELSIF NOT "IX_HBW_SwitchCantileverFront_I5" AND "IX_HBW_SwitchCantileverBack_I6" THEN
                   "QX_HBW_M4_CantileverBackward_Q8" := FALSE;
                   "QX_HBW_M4_CantileverForward_Q7" := FALSE;
                   #li_StepCase := 20;
               END_IF;

           20:  // Set Positioning activ?
               IF "gtyp_HBW".x_Start_Park_Position AND NOT "gtyp_HBW".x_Park_Position_Reached THEN
                   "gtyp_HBW".Horizontal_Axis.x_Start_Positioning := FALSE;
                   "gtyp_HBW".Vertical_Axis.x_Start_Positioning := FALSE;
                   "gtyp_HBW".Horizontal_Axis.x_Reference := FALSE;
                   "gtyp_HBW".Vertical_Axis.x_Reference := FALSE;
                   "QX_HBW_M4_CantileverBackward_Q8" := FALSE;
                   "QX_HBW_M4_CantileverForward_Q7" := FALSE;
                   #li_StepCase := 30;
               END_IF;

           30: // homing vertical axis
               "gtyp_HBW".Vertical_Axis.x_Reference := TRUE;

               IF NOT "gtyp_HBW".Vertical_Axis.x_Referenced THEN
                   #li_StepCase := 40;
               END_IF;

           40: // homed vertical axis
               IF "gtyp_HBW".Vertical_Axis.x_Referenced THEN
                   "gtyp_HBW".Vertical_Axis.x_Reference := FALSE;
                   #li_StepCase := 50;
               END_IF;

           50: // homing horizontal axis
               "gtyp_HBW".Horizontal_Axis.x_Reference := TRUE;

               IF NOT "gtyp_HBW".Horizontal_Axis.x_Referenced THEN
                   #li_StepCase := 60;
               END_IF;

           60: // homed horizontal axis
               IF "gtyp_HBW".Horizontal_Axis.x_Referenced THEN
                   "gtyp_HBW".Horizontal_Axis.x_Reference := FALSE;
                   #li_StepCase := 70;
               END_IF;

           70: // Position horizontal Axis
               "gtyp_HBW".Horizontal_Axis.di_Target_Position := "gtyp_HBW".di_Pos_Park_Horizontal;
               "gtyp_HBW".Horizontal_Axis.x_Start_Positioning := TRUE;

               IF ("gtyp_HBW".Horizontal_Axis.di_Actual_Position <= ("gtyp_HBW".di_Pos_Park_Horizontal + "gtyp_HBW".Horizontal_Axis.Config.di_Pos_Window))
                   AND ("gtyp_HBW".Horizontal_Axis.di_Actual_Position >= ("gtyp_HBW".di_Pos_Park_Horizontal - "gtyp_HBW".Horizontal_Axis.Config.di_Pos_Window))
                   AND "gtyp_HBW".Horizontal_Axis.x_Position_Reached THEN
                   "gtyp_HBW".Horizontal_Axis.x_Start_Positioning := FALSE;
                   #li_StepCase := 80;
               END_IF;

           80: // Position vertical Axis
               "gtyp_HBW".Vertical_Axis.di_Target_Position := "gtyp_HBW".di_Pos_Park_Vertical;
               "gtyp_HBW".Vertical_Axis.x_Start_Positioning := TRUE;

               IF ("gtyp_HBW".Vertical_Axis.di_Actual_Position <= ("gtyp_HBW".di_Pos_Park_Vertical + "gtyp_HBW".Vertical_Axis.Config.di_Pos_Window))
                   AND ("gtyp_HBW".Vertical_Axis.di_Actual_Position >= ("gtyp_HBW".di_Pos_Park_Vertical - "gtyp_HBW".Vertical_Axis.Config.di_Pos_Window))
                   AND "gtyp_HBW".Vertical_Axis.x_Position_Reached THEN
                   "gtyp_HBW".Vertical_Axis.x_Start_Positioning := FALSE;
                   #li_StepCase := 90;
               END_IF;

           90: // Deciding which doing
               "gtyp_HBW".x_Park_Position_Reached := TRUE;


               // Statement section ELSE    
           ELSE
               ;
       END_CASE;

   ELSE
       #lx_Init := TRUE;
   END_IF;
END_FUNCTION_BLOCK

FUNCTION_BLOCK "FB_Axis_Auto"   // FB41, SCL
TITLE = Functionblock Axis
{ S7_Optimized_Access := 'TRUE' }
AUTHOR : A.Schaefer
VERSION : 0.0
   VAR_INPUT
      ini_Axis : Int;
      indi_Increment : DInt;
      inx_Ref_Switch : Bool;
      inx_Start_Positioning : Bool;
      inx_Referencing : Bool;
      ini_PWM : Int;
      indi_Target_Position : DInt;
   END_VAR
   VAR_OUTPUT
      outx_Referenced : Bool;
      outx_Position_Reached : Bool;
      outx_Motor_Pos : Bool;
      outx_Motor_Neg : Bool;
      outi_Motor_PWM : Int;
      outdi_Actual_Position : DInt;
   END_VAR
   VAR_IN_OUT
      inouttyp_Config : "typ_Axis_Data";
      inouttyp_Setup : "typ_SetupAxis";
   END_VAR
   VAR
      li_StepCaseSetup : Int;
      li_StepCase : Int;
      lx_Init : Bool;
      lx_Motor_Neg : Bool;
      lx_Motor_Pos : Bool;
      lx_Start_TON_Wait : Bool;
      li_PWM : Int;
      ldi_ValueStep : DInt;
      ldi_Actual_Position : DInt;
      ldi_Actual_Position_Old : DInt;
      lfb_R_Trig_Setup : R_TRIG;
      lfb_R_Trig_Referencing : R_TRIG;
      lfb_TON_Wait : TON_TIME;
   END_VAR
   VAR_TEMP
      ti_Target_PWM : Int;
   END_VAR
   VAR CONSTANT
      ci_Min_PWM : Int := 400;
      ci_Max_PWM : Int := 900;
      ci_Acceleration : Int := 7;
   END_VAR
BEGIN
   IF #lx_Init THEN

       // rising edge set up axis
       #lfb_R_Trig_Setup(CLK := #inouttyp_Setup.x_Setup_Activ);

       //Reload when switching to set up
       IF #lfb_R_Trig_Setup.Q THEN
           #inouttyp_Setup.di_LoopValue := #inouttyp_Config.di_Loop_Value;
           #inouttyp_Setup.di_Ref_Pos :=
           #inouttyp_Setup.di_Actual_Ref_Pos := #inouttyp_Config.di_Ref_Pos;
           #inouttyp_Setup.di_Soft_End_Pos_Neg :=
           #inouttyp_Setup.di_Actual_Soft_End_Pos_Neg := #inouttyp_Config.di_Neg_Soft_Switch;
           #inouttyp_Setup.di_Soft_End_Pos_Pos :=
           #inouttyp_Setup.di_Actual_Soft_End_Pos_Pos := #inouttyp_Config.di_Pos_Soft_Switch;
           #inouttyp_Setup.i_PWM := #ini_PWM;
           #inouttyp_Setup.x_Approach_Ref_Pos := FALSE;
           #inouttyp_Setup.x_Approach_Target_Pos := FALSE;
           #inouttyp_Setup.x_Axis_Neg := FALSE;
           #inouttyp_Setup.x_Axis_Pos := FALSE;
           #inouttyp_Setup.x_Set_Ref_Pos := FALSE;
           #inouttyp_Setup.x_Set_Soft_End_Pos := FALSE;
       END_IF;

       #ldi_Actual_Position := #indi_Increment;

       //rising edge referencing
       #lfb_R_Trig_Referencing(CLK := #inx_Referencing);

       //waiting period
       #lfb_TON_Wait(IN := #lx_Start_TON_Wait,
                     PT := T#200ms);

       (**********************************)
       (******   set up step chain   *****)
       (**********************************)
       IF #inouttyp_Setup.i_AxisSelection = #ini_Axis AND #inouttyp_Setup.x_Setup_Activ THEN
           IF #inouttyp_Setup.x_Approach_Ref_Pos THEN
               #inouttyp_Setup.i_Function := 10;
           END_IF;

           CASE #inouttyp_Setup.i_Function OF

               0:  // automatic
                   #ldi_Actual_Position_Old := 0;
                   #inouttyp_Setup.x_Approach_Ref_Pos := FALSE;
                   #lx_Start_TON_Wait := FALSE;

               10: // homing
                   IF #inouttyp_Setup.x_Approach_Ref_Pos THEN
                       IF NOT #inx_Ref_Switch THEN
                           #lx_Motor_Neg := TRUE;
                           #lx_Motor_Pos := FALSE;
                           #outx_Referenced := FALSE;
                       END_IF;

                       IF #inx_Ref_Switch THEN
                           #lx_Motor_Neg := TRUE;
                           #lx_Motor_Pos := TRUE;

                           IF #ldi_Actual_Position = #inouttyp_Config.di_Ref_Pos THEN
                               #inouttyp_Setup.x_Approach_Ref_Pos := FALSE;
                               #lx_Motor_Neg := FALSE;
                               #lx_Motor_Pos := FALSE;
                               #outx_Referenced := TRUE;
                           END_IF;
                       END_IF;
                   END_IF;

               20:  // tap
                   #lx_Motor_Neg := #inouttyp_Setup.x_Axis_Neg AND NOT #inx_Ref_Switch AND NOT (#ldi_Actual_Position <= #inouttyp_Setup.di_Soft_End_Pos_Neg);
                   #lx_Motor_Pos := #inouttyp_Setup.x_Axis_Pos AND NOT #lx_Motor_Neg AND NOT (#ldi_Actual_Position >= #inouttyp_Setup.di_Soft_End_Pos_Pos);

               30:  // tap with increment
                   #ldi_Actual_Position_Old := #ldi_Actual_Position;

                   // positiv
                   IF #inouttyp_Setup.x_Axis_Pos AND NOT ((#ldi_Actual_Position + #inouttyp_Setup.w_Increment + #inouttyp_Setup.di_LoopValue) >= #inouttyp_Setup.di_Soft_End_Pos_Pos) THEN
                       #lx_Motor_Neg := FALSE;
                       #lx_Motor_Pos := TRUE;
                       #ldi_ValueStep := #ldi_Actual_Position_Old + #inouttyp_Setup.w_Increment;

                       // without loop
                       IF (#inouttyp_Setup.di_LoopValue = 0) THEN
                           #inouttyp_Setup.i_Function := 36;
                       ELSE
                           #inouttyp_Setup.i_Function := 31;
                       END_IF;
                       // negativ
                   ELSIF #inouttyp_Setup.x_Axis_Neg AND NOT ((#ldi_Actual_Position - #inouttyp_Setup.w_Increment) <= #inouttyp_Config.di_Neg_Soft_Switch) THEN
                       #lx_Motor_Neg := TRUE;
                       #lx_Motor_Pos := FALSE;
                       #ldi_ValueStep := #ldi_Actual_Position_Old - #inouttyp_Setup.w_Increment;
                       #inouttyp_Setup.i_Function := 34;
                   END_IF;

               31: // with loop
                   IF ((#ldi_Actual_Position >= (#ldi_ValueStep + #inouttyp_Setup.di_LoopValue - #inouttyp_Config.di_Pos_Window)) = 0) THEN
                       #lx_Motor_Neg := TRUE;
                       #lx_Motor_Pos := TRUE;
                       #inouttyp_Setup.i_Function := 32;
                   END_IF;

               32: // wait sequence
                   #lx_Start_TON_Wait := TRUE;

                   IF #lfb_TON_Wait.Q THEN
                       #lx_Motor_Neg := FALSE;
                       #lx_Motor_Pos := FALSE;
                       #lx_Start_TON_Wait := FALSE;
                       #inouttyp_Setup.i_Function := 33;
                   END_IF;

               33: // change direction
                   #lx_Motor_Neg := TRUE;
                   #lx_Motor_Pos := FALSE;
                   #inouttyp_Setup.i_Function := 34;

               34: // position reached negativ
                   IF (#ldi_Actual_Position <= (#ldi_ValueStep + #inouttyp_Config.di_Pos_Window))
                       AND (#ldi_Actual_Position >= (#ldi_ValueStep - #inouttyp_Config.di_Pos_Window)) THEN
                       #lx_Motor_Neg := TRUE;
                       #lx_Motor_Pos := TRUE;
                       #inouttyp_Setup.i_Function := 35;
                   END_IF;

               35: // wait sequence
                   #lx_Start_TON_Wait := TRUE;

                   IF #lfb_TON_Wait.Q THEN
                       #lx_Motor_Neg := FALSE;
                       #lx_Motor_Pos := FALSE;
                       #lx_Start_TON_Wait := FALSE;
                       #inouttyp_Setup.x_Axis_Neg := FALSE;
                       #inouttyp_Setup.x_Axis_Pos := FALSE;
                       #inouttyp_Setup.i_Function := 30;
                   END_IF;


               36: // position reached positiv
                   IF (#ldi_Actual_Position <= (#ldi_ValueStep + #inouttyp_Config.di_Pos_Window))
                       AND (#ldi_Actual_Position >= (#ldi_ValueStep - #inouttyp_Config.di_Pos_Window)) THEN
                       #lx_Motor_Neg := TRUE;
                       #lx_Motor_Pos := TRUE;
                       #inouttyp_Setup.i_Function := 37;
                   END_IF;

               37: // wait sequence
                   #lx_Start_TON_Wait := TRUE;

                   IF #lfb_TON_Wait.Q THEN
                       #lx_Motor_Neg := FALSE;
                       #lx_Motor_Pos := FALSE;
                       #lx_Start_TON_Wait := FALSE;
                       #inouttyp_Setup.x_Axis_Neg := FALSE;
                       #inouttyp_Setup.x_Axis_Pos := FALSE;
                       #inouttyp_Setup.i_Function := 30;
                   END_IF;

               40: // approach position
                   IF #inouttyp_Setup.x_Approach_Target_Pos THEN
                       // positiv
                       IF (#inouttyp_Setup.di_Target_Position > #ldi_Actual_Position) AND NOT ((#inouttyp_Setup.di_Target_Position + #inouttyp_Setup.di_LoopValue) >= #inouttyp_Setup.di_Soft_End_Pos_Pos) THEN
                           #lx_Motor_Neg := FALSE;
                           #lx_Motor_Pos := TRUE;
                           // without loop
                           IF (#inouttyp_Setup.di_LoopValue = 0) THEN
                               #inouttyp_Setup.i_Function := 46;
                           ELSE
                               #inouttyp_Setup.i_Function := 41;
                           END_IF;
                           // negativ
                       ELSIF ((#inouttyp_Setup.di_Target_Position < #ldi_Actual_Position) AND NOT (#inouttyp_Setup.di_Target_Position <= #inouttyp_Config.di_Neg_Soft_Switch)) THEN
                           #lx_Motor_Neg := TRUE;
                           #lx_Motor_Pos := FALSE;
                           #inouttyp_Setup.i_Function := 44;
                       ELSIF (#inouttyp_Setup.di_Target_Position = #ldi_Actual_Position) THEN
                           #inouttyp_Setup.i_Function := 46;
                       END_IF;

                   END_IF;

               41: // with loop
                   IF (#ldi_Actual_Position >= (#inouttyp_Setup.di_Target_Position + #inouttyp_Setup.di_LoopValue - #inouttyp_Config.di_Pos_Window)) THEN
                       #lx_Motor_Neg := TRUE;
                       #lx_Motor_Pos := TRUE;
                       #inouttyp_Setup.i_Function := 42;
                   END_IF;

               42: // wait sequence
                   #lx_Start_TON_Wait := TRUE;

                   IF #lfb_TON_Wait.Q THEN
                       #lx_Motor_Neg := FALSE;
                       #lx_Motor_Pos := FALSE;
                       #lx_Start_TON_Wait := FALSE;
                       #inouttyp_Setup.i_Function := 43;
                   END_IF;

               43: // change direction
                   #lx_Motor_Neg := TRUE;
                   #lx_Motor_Pos := FALSE;
                   #inouttyp_Setup.i_Function := 44;

               44: // position reached negativ
                   IF (#ldi_Actual_Position <= (#inouttyp_Setup.di_Target_Position + #inouttyp_Config.di_Pos_Window))
                       AND (#ldi_Actual_Position >= (#inouttyp_Setup.di_Target_Position - #inouttyp_Config.di_Pos_Window)) THEN
                       #lx_Motor_Neg := TRUE;
                       #lx_Motor_Pos := TRUE;
                       #inouttyp_Setup.i_Function := 45;
                   END_IF;

               45: // wait sequence
                   #lx_Start_TON_Wait := TRUE;

                   IF #lfb_TON_Wait.Q THEN
                       #lx_Motor_Neg := FALSE;
                       #lx_Motor_Pos := FALSE;
                       #lx_Start_TON_Wait := FALSE;
                       #inouttyp_Setup.x_Axis_Neg := FALSE;
                       #inouttyp_Setup.x_Axis_Pos := FALSE;
                       #inouttyp_Setup.i_Function := 40;
                   END_IF;

               46: //  position reached positiv
                   IF (#ldi_Actual_Position <= (#inouttyp_Setup.di_Target_Position + #inouttyp_Config.di_Pos_Window))
                       AND (#ldi_Actual_Position >= (#inouttyp_Setup.di_Target_Position - #inouttyp_Config.di_Pos_Window)) THEN
                       #lx_Motor_Neg := TRUE;
                       #lx_Motor_Pos := TRUE;
                       #inouttyp_Setup.i_Function := 47;
                   END_IF;

               47:  // wait sequence
                   #lx_Start_TON_Wait := TRUE;

                   IF #lfb_TON_Wait.Q THEN
                       #lx_Motor_Neg := FALSE;
                       #lx_Motor_Pos := FALSE;
                       #lx_Start_TON_Wait := FALSE;
                       #inouttyp_Setup.x_Approach_Target_Pos := FALSE;
                       #inouttyp_Setup.i_Function := 40;
                   END_IF;
               ELSE  // Statement section ELSE
                   ;
           END_CASE;

           // set reference point
           IF #inouttyp_Setup.x_Set_Ref_Pos THEN
               #inouttyp_Setup.di_Actual_Ref_Pos :=
               #inouttyp_Config.di_Ref_Pos := #inouttyp_Setup.di_Ref_Pos;
               #inouttyp_Setup.x_Set_Ref_Pos := FALSE;
           END_IF;

           // set software end position
           IF #inouttyp_Setup.x_Set_Soft_End_Pos THEN
               #inouttyp_Setup.di_Actual_Soft_End_Pos_Neg :=
               #inouttyp_Config.di_Neg_Soft_Switch := #inouttyp_Setup.di_Soft_End_Pos_Neg;
               #inouttyp_Setup.di_Actual_Soft_End_Pos_Pos :=
               #inouttyp_Config.di_Pos_Soft_Switch := #inouttyp_Setup.di_Soft_End_Pos_Pos;
               #inouttyp_Setup.x_Set_Soft_End_Pos := FALSE;
           END_IF;

           // reload PWM
           #li_PWM := #inouttyp_Setup.i_PWM;

           // reload actual position
           #inouttyp_Setup.di_ActualPosition := #ldi_Actual_Position;

           (************************************)
           (******   position step chain   *****)
           (************************************)
       ELSIF NOT #inouttyp_Setup.x_Setup_Activ THEN

           // rising edge set up axis
           IF #lfb_R_Trig_Referencing.Q THEN
               #li_StepCase := 0;
           END_IF;

           CASE #li_StepCase OF

               0:  // init
                   #lx_Start_TON_Wait := FALSE;

                   IF #inx_Referencing THEN
                       #li_StepCase := 10;
                       #outx_Position_Reached := FALSE;
                       #outx_Referenced := FALSE;
                   ELSIF #inx_Start_Positioning THEN
                       #li_StepCase := 20;
                       #outx_Position_Reached := FALSE;
                   END_IF;

               10: // homing
                   IF NOT #inx_Ref_Switch THEN
                       #lx_Motor_Neg := TRUE;
                       #lx_Motor_Pos := FALSE;
                   END_IF;

                   IF #inx_Ref_Switch THEN
                       #lx_Motor_Neg := TRUE;
                       #lx_Motor_Pos := TRUE;

                       IF #inx_Ref_Switch THEN
                           IF #ldi_Actual_Position = #inouttyp_Config.di_Ref_Pos THEN
                               #lx_Motor_Neg := FALSE;
                               #lx_Motor_Pos := FALSE;
                               #outx_Referenced := TRUE;
                               #li_StepCase := 11;
                           END_IF;
                       END_IF;
                   END_IF;

               11: // wait not referencing
                   IF NOT #inx_Referencing THEN
                       #li_StepCase := 0;
                   END_IF;

               20: // approach position
                   // positiv
                   IF (#indi_Target_Position > #ldi_Actual_Position) AND NOT ((#indi_Target_Position + #inouttyp_Config.di_Loop_Value) >= #inouttyp_Config.di_Pos_Soft_Switch) THEN
                       #lx_Motor_Neg := FALSE;
                       #lx_Motor_Pos := TRUE;
                       //without loop
                       IF (#inouttyp_Config.di_Loop_Value = 0) THEN
                           #li_StepCase := 26;
                       ELSE
                           #li_StepCase := 21;
                       END_IF;
                       // negativ
                   ELSIF ((#indi_Target_Position < #ldi_Actual_Position) AND NOT (#indi_Target_Position <= #inouttyp_Config.di_Neg_Soft_Switch)) THEN
                       #lx_Motor_Neg := TRUE;
                       #lx_Motor_Pos := FALSE;
                       #li_StepCase := 24;
                   ELSIF (#indi_Target_Position = #ldi_Actual_Position) THEN
                       #li_StepCase := 26;
                   END_IF;

               21: // with loop
                   IF (#ldi_Actual_Position >= (#indi_Target_Position + #inouttyp_Config.di_Loop_Value - #inouttyp_Config.di_Pos_Window)) THEN
                       #lx_Motor_Neg := TRUE;
                       #lx_Motor_Pos := TRUE;
                       #li_StepCase := 22;
                   END_IF;

               22: // wait sequence
                   #lx_Start_TON_Wait := TRUE;

                   IF #lfb_TON_Wait.Q THEN
                       #lx_Motor_Neg := FALSE;
                       #lx_Motor_Pos := FALSE;
                       #lx_Start_TON_Wait := FALSE;
                       #inouttyp_Setup.i_Function := 23;
                   END_IF;

               23: // change direction
                   #lx_Motor_Neg := TRUE;
                   #lx_Motor_Pos := FALSE;
                   #li_StepCase := 24;

               24: // position reached negativ
                   IF (#ldi_Actual_Position <= (#indi_Target_Position + #inouttyp_Config.di_Pos_Window))
                       AND (#ldi_Actual_Position >= (#indi_Target_Position - #inouttyp_Config.di_Pos_Window)) THEN
                       #lx_Motor_Neg := TRUE;
                       #lx_Motor_Pos := TRUE;
                       #li_StepCase := 25;
                   END_IF;

               25: // wait sequence
                   #lx_Start_TON_Wait := TRUE;

                   IF #lfb_TON_Wait.Q THEN
                       #lx_Motor_Neg := FALSE;
                       #lx_Motor_Pos := FALSE;
                       #lx_Start_TON_Wait := FALSE;
                       #outx_Position_Reached := TRUE;
                       #li_StepCase := 28;
                   END_IF;

               26: // position reached positiv
                   IF (#ldi_Actual_Position <= (#indi_Target_Position + #inouttyp_Config.di_Pos_Window))
                       AND (#ldi_Actual_Position >= (#indi_Target_Position - #inouttyp_Config.di_Pos_Window)) THEN
                       #lx_Motor_Neg := TRUE;
                       #lx_Motor_Pos := TRUE;
                       #li_StepCase := 27;
                   END_IF;

               27: // wait sequence
                   #lx_Start_TON_Wait := TRUE;

                   IF #lfb_TON_Wait.Q THEN
                       #lx_Motor_Neg := FALSE;
                       #lx_Motor_Pos := FALSE;
                       #lx_Start_TON_Wait := FALSE;
                       #outx_Position_Reached := TRUE;
                       #li_StepCase := 28;
                   END_IF;

               28: // wait not start positioning
                   IF NOT #inx_Start_Positioning THEN
                       #li_StepCase := 0;
                   END_IF;
                   // statement section ELSE    
               ELSE
                   ;
           END_CASE;

           IF #ini_PWM = -1 THEN
               //Automatically calculate the PWM value
               IF #inx_Referencing THEN
                   //If the position is less then 0 slow the axis down
                   IF #ldi_Actual_Position <= 0 THEN
                       //If the position is less than 0, position is likely not known, so slow down
                       #li_PWM := #ci_Min_PWM;
                   ELSE
                       //When referencing the target position is 0, so the position can be used as speed
                       #ti_Target_PWM := DINT_TO_INT(MIN_DINT(IN1 := #ldi_Actual_Position + #ci_Min_PWM, IN2 := #ci_Max_PWM));
                       //If the desired speed is greater than current, accelerate
                       IF #ti_Target_PWM > #li_PWM THEN
                           #li_PWM := #li_PWM + #ci_Acceleration;
                       ELSE
                           #li_PWM := #ti_Target_PWM;
                       END_IF;
                   END_IF;
               ELSE
                   //When regular moving, use the distance as PWM
                   #ti_Target_PWM := DINT_TO_INT(MIN_DINT(IN1 := ABS_DINT(#ldi_Actual_Position - #indi_Target_Position) + #ci_Min_PWM, IN2 := #ci_Max_PWM));
                   //If the desired speed is greater than current, accelerate
                   IF #ti_Target_PWM > #li_PWM THEN
                       #li_PWM := #li_PWM + #ci_Acceleration;
                   ELSE
                       #li_PWM := #ti_Target_PWM;
                   END_IF;
               END_IF;
           ELSE
               #li_PWM := #ini_PWM;
           END_IF;
       END_IF;

       // reload outputs
       #outx_Motor_Neg := #lx_Motor_Neg;
       #outx_Motor_Pos := #lx_Motor_Pos;
       #outi_Motor_PWM := #li_PWM;
       #outdi_Actual_Position := #ldi_Actual_Position;

   ELSE
       #lx_Init := TRUE;
   END_IF;
END_FUNCTION_BLOCK

FUNCTION "FC_Scale_linear" : Real   // FC1, SCL
TITLE = Function scale linear
{ S7_Optimized_Access := 'TRUE' }
AUTHOR : A.Schaefer
VERSION : 0.0
   VAR_INPUT
      inr_Y1 : Real;   // Initial scaling value for Y (INPUT)
      inr_Y2 : Real;   // Scaling end value for Y (INPUT)
      inr_X1 : Real;   // Initial scaling value for X (INPUT)
      inr_X2 : Real;   // Scaling end value for X (INPUT)
      inr_X : Real;   // Value to be scaled
   END_VAR
   VAR_TEMP
      lr_y_delta : Real;   // Temp delta y
      lr_x_delta : Real;   // Temp delta x
      lr_m : Real;   // Temp gradient m
   END_VAR
BEGIN
   (********************************************************)
   (* FC for linear scaling. Line function  y=m*(x-x1)+y1  *)
   (********************************************************)

   #lr_y_delta := (#inr_Y2 - #inr_Y1);
   #lr_x_delta := (#inr_X2 - #inr_X1);

   IF #lr_y_delta <> 0 AND #lr_x_delta <> 0 THEN
       #lr_m := (#lr_y_delta / #lr_x_delta);
       #FC_Scale_linear := (#lr_m * (#inr_X - #inr_X1)) + #inr_Y1;
   ELSE
       #FC_Scale_linear := 0;
   END_IF;
END_FUNCTION

ORGANIZATION_BLOCK "Main"   // OB1, SCL, ProgramCycle
TITLE = "Main Program Sweep (Cycle)"
{ S7_Optimized_Access := 'TRUE' }
AUTHOR : A.Schaefer
VERSION : 0.0
   VAR_INPUT
      Initial_Call : Bool;   // Initial call of this OB
      Remanence : Bool;   // =True, if remanent data are available
   END_VAR
BEGIN
   // current cycle Time OB30
   "RT_INFO_scl_OB30".mode := 1;
   "RT_INFO_scl_OB30".obNbr := 30;
   "RT_INFO_scl_OB30".returnValue := RT_INFO(MODE := "RT_INFO_scl_OB30".mode,
                                             OB := "RT_INFO_scl_OB30".obNbr,
                                             INFO := "RT_INFO_scl_OB30".infoData);

   // current cycle Time OB1
   "RT_INFO_scl_OB1".mode := 1;
   "RT_INFO_scl_OB1".obNbr := 1;
   "RT_INFO_scl_OB1".returnValue := RT_INFO(MODE := "RT_INFO_scl_OB1".mode,
                                            OB := "RT_INFO_scl_OB1".obNbr,
                                            INFO := "RT_INFO_scl_OB1".infoData);

   // sources SSC
   "PRG_SSC_Ablauf_DB"();
   "PRG_SSC_Set_Positioning_DB"();
   "PRG_SSC_Set_Park_Position_DB"();
   "PRG_SSC_Calibration_Color_DB"();
   "PRG_SSC_Axis_Vertical_DB"();
   "PRG_SSC_Axis_Horizontal_DB"();
   "PRG_SSC_Light_DB"();

   // sources VGR
   "PRG_VGR_Ablauf_DB"();
   "PRG_VGR_Set_Positioning_DB"();
   "PRG_VGR_Set_Park_Position_DB"();
   "PRG_VGR_Axis_horizontal_DB"();
   "PRG_VGR_Axis_vertical_DB"();
   "PRG_VGR_Axis_rotate_DB"();
   "PRG_NFC_DB"();

   // sources HBW
   "PRG_HBW_Ablauf_DB"();
   "PRG_HBW_Set_Positioning_DB"();
   "PRG_HBW_Set_Park_Position_DB"();
   "PRG_HBW_Axis_Vertical_DB"();
   "PRG_HBW_Axis_Horizontal_DB"();

   // sources MPO
   "PRG_MPO_Ablauf_DB"();
   "PRG_MPO_Set_Park_Position_DB"();

   // sources SLD
   "PRG_SLD_Ablauf_DB"();
   "PRG_SLD_Calibration_Color_DB"();
   "PRG_SLD_Set_Counter_Values_DB"();

   // sources input/output
   "PRG_DSI_Status_DB"();
   "PRG_DSO_Status_DB"();

   // sources dashboard
   "PRG_Order_DB"();
   "PRG_Acknowledge_DB"();

   // communication 
   "Copy_Simulation_Variables_DB"();
END_ORGANIZATION_BLOCK

ORGANIZATION_BLOCK "Cyclic interrupt"   // OB30, SCL, CyclicInterrupt
TITLE = Cyclic interrupt
{ S7_Optimized_Access := 'TRUE' }
AUTHOR : A.Schaefer
VERSION : 0.0
   VAR_INPUT
      Initial_Call : Bool;   // Initial call of this OB
      Event_Count : Int;   // Events discarded
   END_VAR
   VAR_TEMP
      li_Return_LDT : Int;
   END_VAR
BEGIN

   "PRG_SSC_Axis_Horizontal_Act_Pos_DB"();
   "PRG_SSC_Axis_Vertical_Act_Pos_DB"();

   "PRG_HBW_Axis_Horizontal_Act_Pos_DB"();
   "PRG_HBW_Axis_Vertical_Act_Pos_DB"();

   "PRG_VGR_Axis_horizontal_Act_Pos_DB"();
   "PRG_VGR_Axis_vertical_Act_Pos_DB"();
   "PRG_VGR_Axis_rotate_Act_Pos_DB"();
END_ORGANIZATION_BLOCK